PROGRAM PG_Wind
VAR
	FB_Wind_0: FB_Wind;
	INT_TRIG_0: INT_TRIG;
	FB_DataHistory_Real_0: FB_DataHistory_Real;
	R_TRIG_0: R_TRIG;
END_VAR
VAR // added by the converter: edge detectors and wires of the graphical bodies
    _w1 : BOOL;
END_VAR

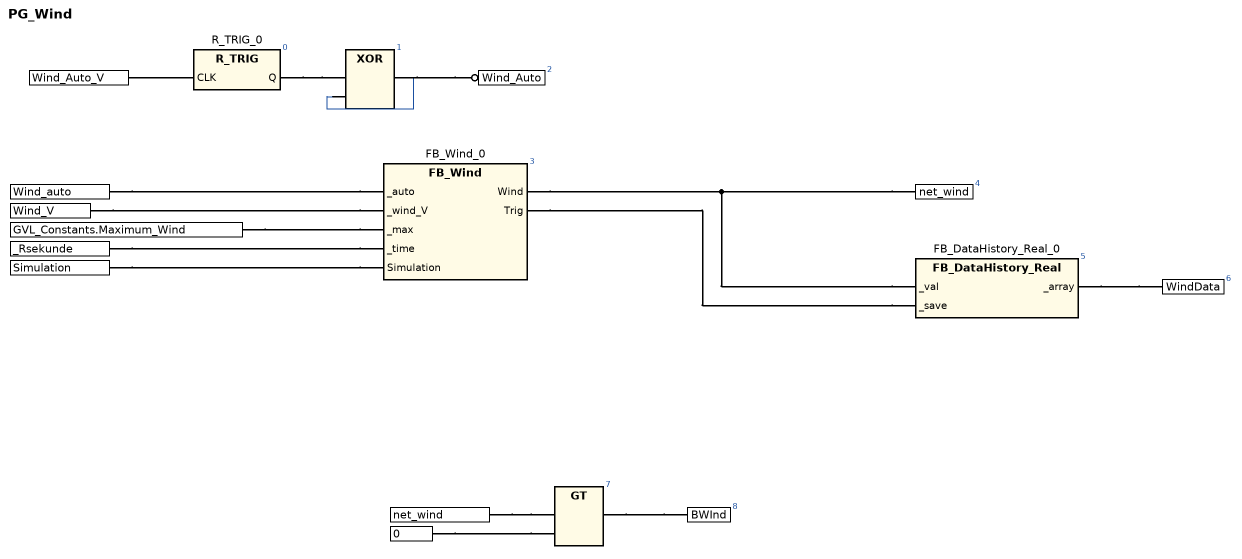
R_TRIG_0(CLK := Wind_Auto_V); // R_TRIG
_w1 := R_TRIG_0.Q XOR _w1;
Wind_Auto := NOT _w1;
FB_Wind_0(
    _auto := Wind_auto,
    _wind_V := Wind_V,
    _max := GVL_Constants.Maximum_Wind,
    _time := _Rsekunde,
    Simulation := Simulation); // FB_Wind
net_wind := FB_Wind_0.Wind;
FB_DataHistory_Real_0(_val := FB_Wind_0.Wind, _save := FB_Wind_0.Trig); // FB_DataHistory_Real
WindData := FB_DataHistory_Real_0._array;
BWInd := net_wind > 0;

END_PROGRAM

(* stored: Version 1.1.0.1, ProductVersion 3.1.4018.5
   POU PG_Wind: Id {ce04e43a-2e30-445e-840d-2667f09900af}, SpecialFunc None *)
